{attribute addProperty BoxType "EL3312-0000-0018"}
{attribute addProperty Id "StatusAT %I*Status_34730D861621ValueAT %I*INT16217"}
{attribute addProperty CRC "4291910102"}
{attribute addProperty SizeInBites "32"}
{attribute addProperty SizeInBytes "4"}
TYPE TC_Inputs_Channel_FFD159D6 :
STRUCT
	{attribute addProperty Name "Status"}
	Status AT %I* : Status_34730D86;
	{attribute addProperty Name "Value"}
	Value AT %I* : INT;
END_STRUCT
END_TYPE

(* stored: Version 1.2.0.0, ProductVersion 3.1.4024.9
   DUT TC_Inputs_Channel_FFD159D6: Id {8a1bb756-d9a8-4cf7-a28f-a7656a782250} *)
